TYPE us_LOG_VIEWPORT :
STRUCT
	LINE_ARRAY : ARRAY [1..40] OF INT;
	COUNT : INT; (* Anzahl der sichtbaren Nachtrichten *)
	UPDATE_COUNT : UINT; (* Updatezähler *)
	MOVE_TO_X : INT; (* Steuerung der Nachrichtenanzeige *)
	UPDATE : BOOL; (* Daten wurden geändert -> neuzeichnen *)
END_STRUCT
END_TYPE

(* stored: Version 1.1.0.1, ProductVersion 3.1.4024.4
   DUT us_LOG_VIEWPORT: Id {f1df9103-992a-48cc-8638-64ccb26961e0} *)
